	            IF #Return = TRUE THEN
	                IF #REC._FgDemArr = TRUE THEN
	                    #REC.Dial_Def.Num_Def_Etape := 1;
	                    #REC.Dial_Def.Index_Defaut := "Dialog_Defaut"(Fg_Base := #fgbase, Msg_Defaut := 'Arret immediat',
	                                                                  Type_Defaut := 2,
	                                                                  Automatisme := #REC.RecCommun.CommunGeneral._Autom,
	                                                                  Num_Lot := #REC._Ptzs._NoLot,
	                                                                  Origine_Defaut := 'Pas daction durant la suspension',
	                                                                  Libelle_Origine := 'Confirmez vous larret',
	                                                                  Acq1 := 'Confirmez',
	                                                                  Acq2 := 'Annuler',
	                                                                  Acq3 := '',
	                                                                  Acq4 := '',
	                                                                  Acq5 := '',
	                                                                  Acq6 := '',
	                                                                  Acq7 := '',
	                                                                  Acq8 := '',
	                                                                  Acq_Choisi := -1,
	                                                                  Date_Arrivee := #REC._TpsPicke);
	                    #REC.RecCommun.CommunGeneral._Etp := #Etape_Attente_RepDial;
	                    RETURN;
	                ELSE
	                    #Ret := "Arr_Imm_Circuit"(#REC._PtCir);
	                    #REC.Dial_Def.Reponse_Def := '';
	                    #REC._FgConfArret := TRUE;
	                    (* #Ret := "Arr_Imm_Circuit"(#REC._PtCir);
	                    #REC.RecCommun.CommunGeneral._Etp :=  #Etape_fin_lot; *)
	                    RETURN;
	                END_IF;
	            END_IF;
	        SUSPENSION_DEF1:
	            //======================== Traitement des reponses pour le defaut1 Etape Suspension  ====================================//
	            IF #REC.Dial_Def.Reponse_Def = 'Confirmez' THEN
	                #Ret := "Arr_Imm_Circuit"(#REC._PtCir);
	                #REC.Dial_Def.Reponse_Def := '';
	                #REC._FgConfArret := TRUE;
	                // #REC.RecCommun.CommunGeneral._Etp :=  #Etape_fin_lot;
	                RETURN;
	            END_IF;
	            IF #REC.Dial_Def.Reponse_Def = 'Annuler' THEN
	                //Renitialiser la temporisation pour refaire le test
	                #Ret_RD_Sys_T := RD_SYS_T(#REC._TpsPicke);
	                #REC.Dial_Def.Reponse_Def := '';
	                RETURN;
	            END_IF;
	            //======================================  Fin traitement====================================//
	            (* //pas de dialogue pour Confirmez l'arret
	            IF #Return AND #REC._FgDemArr = FALSE THEN
	                #Ret := "Arr_Imm_Circuit"(#REC._PtCir);
	                #REC.Dial_Def.Reponse_Def := '';
	                #REC._FgConfArret := TRUE;
	                (* #Ret := "Arr_Imm_Circuit"(#REC._PtCir);
	                #REC.RecCommun.CommunGeneral._Etp :=  #Etape_fin_lot; *)
	                RETURN;
	            END_IF; *)
	            IF (#REC._FgArret = TRUE) THEN
	                #REC._Ptzs._QteLot := #REC.RecCommun.CommunGeneral._ParCal._QteTrans;

	                "MAJ_Cumul_Dest"(Dest := "Nom_Mobile"(#REC.RecCommun.CommunGeneral._Ptdest),
	                                 Increment := FALSE,
	                                 DestR := #REC._Ptzs._DestR,
	                                 PARCAL := #REC.RecCommun.CommunGeneral._ParCal);
	                //Fin_Lot_Circuit(_ptCir, _ptCir->Origine.Mobile, _ptCir->Destination.Mobile, pt_zs->QteLot);
	                #REC.RecCommun.CommunGeneral._Etp := #Etape_maj_base;
	                RETURN;
	            END_IF;
	            IF #REC._FgSusp = FALSE THEN
	                //APPEL FCT MARCHE MOB
	                //"DB_BIBLIOTHEQUE".Mobile["DB_BIBLIOTHEQUE".Mobile[#REC._PtCir.Origine].Mob_Suiv[0]].Ord := 0; // Appl fct arrt mob
	                IF NOT #REC._FgConfArret THEN
	                    #Ret := "Dem_Mobile"("DB_BIBLIOTHEQUE".Mobile[#REC._PtCir.Origine].Mob_Suiv[0]);
	                    #REC.RecCommun.CommunGeneral._Etp := #Etape_surveillance;
	                    RETURN;
	                ELSE
	                    #REC.RecCommun.CommunGeneral._Etp := #Etape_prepositionnement;
	                    RETURN;
	                END_IF;




	            END_IF;
	            IF (#REC._FgDemVid = TRUE) THEN
	                //#REC._FgSusp := FALSE;
	                #REC.RecCommun.CommunGeneral._Etp := #Etape_vidange;
	                RETURN;
	            END_IF;


	        END_REGION Traitement cyclique "Suspension"
	        RETURN;
	(*
	 *************************************** *************************************** *************************************** *************************************** *************************************** ***************************************
	                                                                                 ╔════════════════════════════════════╗
	                                                                                 ║        Etape "Test Qte passée"     ║
	                                                                                 ╚════════════════════════════════════╝
	 *************************************** *************************************** *************************************** *************************************** *************************************** ***************************************
	*)
	    #Etape_test_qte_passee:
	        REGION Traitement preliminaire 'Test qte passee'
	            IF (#REC.RecCommun.CommunGeneral._Etp <> #REC.RecCommun.CommunGeneral._EtpPrec) THEN

	                //Memorisation de l'etape encours
	                #REC.RecCommun.CommunGeneral._EtpPrec := #REC.RecCommun.CommunGeneral._Etp;
	                //Reperer le niveau du grafcet
	                #MajNiv := "Maj_Niv"(Num_Zone := #REC.RecCommun.CommunGeneral._NumZone, Num_Tache := #REC.RecCommun.CommunGeneral._Tache, Niveau := "REC_TestQtePassee_Niv");
	                //Nomination l'etape en cours
	                #REC.RecCommun.CommunGeneral._DescEtp := 'Test qte pasee';
	                IF #REC.Dial_Def.Reponse_Def <> '' THEN
	                    CASE #REC.Dial_Def.Num_Def_Etape OF
	                        1:
	                            GOTO TEST_QTE_PASSEE_DEF1;
	                    END_CASE;
	                END_IF;
	                #Ret_RD_Sys_T := RD_SYS_T(#REC._TpsPicke);
	                #REC._DebutMax := #REC._TpsPicke;
	                IF #REC.RecCommun.CommunGeneral._ParCal._DebVolTrans = 0 OR #REC.RecCommun.CommunGeneral._ParCal._DebMasTrans = 0 OR
	                    #REC.RecCommun.CommunGeneral._ParCal._QteTrans = 0 OR #REC._TheoTrans = 0 OR #REC._SeuilTrans = 0
	                    OR #REC._FgTestQtP = FALSE THEN
	                    #REC.RecCommun.CommunGeneral._Etp := #Etape_vidange;
	                    RETURN;
	                END_IF;
	                #REC._FgAbandon := FALSE;
	            END_IF;
	        END_REGION Traitement preliminaire 'Test qte passee'

	        REGION Traitement cyclique "Test qte passee"
	            // mise a jour quantité theorique calculé en zone de suivi
	            #REC._Ptzs._Qte_Rec := #REC.RecCommun.CommunGeneral._ParCal._QteTrans;
	            // mise a jour temps de marche transporteur dans zone de suivi
	            #REC._Ptzs._Tps_Tc := #REC.RecCommun.CommunGeneral._ParCal._TpsTran;
	            //calcul debit massique
	            "Debit_Massique"(SAV := #REC._vitesseFosse,
	                             Densite := #REC._Ptzs._Densite,
	                             PARCAL := #REC.RecCommun.CommunGeneral._ParCal);
	            //test demande d'arret par bouton sur supervision
	            IF #REC._FgArret THEN
	                #REC.RecCommun.CommunGeneral._Etp := #Etape_vidange;
	                RETURN;
	            END_IF;
	            //test demande de vidange par bouton sur supervision
	            IF #REC._FgDemVid THEN
	                #REC.RecCommun.CommunGeneral._Etp := #Etape_vidange;
	                RETURN;
	            END_IF;
	            //test demande de suspension par bouton sur supervision
	            IF #REC._FgSusp THEN
	                #REC.RecCommun.CommunGeneral._Etp := #Etape_suspension;
	                RETURN;
	            END_IF;
	            //teste niveau haut
	            #Ret := "Controle_NH"(TempoAffNH := "TpDefNh", R := #REC);
	            IF #Ret = 1 THEN
	                #REC.RecCommun.CommunGeneral._Etp := #Etape_changement_destination;
	                RETURN;
	            END_IF;
	            //Controle quantité passée
	            IF #REC.RecCommun.CommunGeneral._ParCal._QteTrans >= (#REC._TheoTrans - #REC._SeuilTrans) OR #REC._FgAbandon THEN
	                IF #REC._FgAbandon = FALSE THEN
	                    #REC._Ptzs._Fg_Qte_Passee := TRUE;
	                END_IF;
	                #REC.RecCommun.CommunGeneral._Etp := #Etape_vidange;
	                RETURN;
	            END_IF;
	            //decompte tempo maxi avant dialogue de defaut
	            #Return := "Tempo"(Duree := #REC._TpMaxFPm, Tps_Picke := #REC._DebutMax, Anticip := FALSE, Tps_Passe => #Tps_Passe);
	            IF #Return AND #REC._FgAbandon = false THEN
	                #REC.Dial_Def.Num_Def_Etape := 1;
	                #REC.Dial_Def.Index_Defaut := "Dialog_Defaut"(Fg_Base := #fgbase, Msg_Defaut := 'Perte de matiere',
	                                                              Type_Defaut := 2,
	                                                              Automatisme := #REC.RecCommun.CommunGeneral._Autom,
	                                                              Num_Lot := #REC._Ptzs._NoLot,
	                                                              Origine_Defaut := 'Pas de presence du matiere',
	                                                              Libelle_Origine := 'Pas de presence du matiere',
	                                                              Acq1 := 'Relance',
	                                                              Acq2 := 'Abandon',
	                                                              Acq3 := '',
	                                                              Acq4 := '',
	                                                              Acq5 := '',
	                                                              Acq6 := '',
	                                                              Acq7 := '',
	                                                              Acq8 := '',
	                                                              Acq_Choisi := -1,
	                                                              Date_Arrivee := #REC._TpsPicke);
	                #REC.RecCommun.CommunGeneral._Etp := #Etape_Attente_RepDial;
	                RETURN;
	            END_IF;
	        TEST_QTE_PASSEE_DEF1:
	            //======================== Traitement des reponses pour le defaut1 Etape TEST QTE PASSEE Perte PM  ====================================//
	            IF #REC.Dial_Def.Reponse_Def = 'Relance' THEN //relance
	                #REC._DebutMax := #REC._TpsPicke;
	                #REC.Dial_Def.Reponse_Def := '';
	                RETURN;
	            END_IF;
	            IF #REC.Dial_Def.Reponse_Def = 'Abandon' THEN //abandon
	                #REC._FgAbandon := TRUE;
	                #REC.Dial_Def.Reponse_Def := '';
	                RETURN;
	            END_IF;
	            //======================================  Fin traitement====================================//
	        END_REGION Traitement cyclique "Test qte passee"

	        RETURN;
	(*
	 *************************************** *************************************** *************************************** *************************************** *************************************** ***************************************
	                                                                                 ╔════════════════════════════════════╗
	                                                                                 ║   Etape "Attente Acq nettoyage"    ║
	                                                                                 ╚════════════════════════════════════╝
	 *************************************** *************************************** *************************************** *************************************** *************************************** ***************************************
	*)
	    #Etape_attente_acquit_nettoyage:

	        REGION Traitement preliminaire 'Attente_acquit_nettoyage'
	            IF (#REC.RecCommun.CommunGeneral._Etp <> #REC.RecCommun.CommunGeneral._EtpPrec) THEN
	                //Memorisation de l'etape encours
	                #REC.RecCommun.CommunGeneral._EtpPrec := #REC.RecCommun.CommunGeneral._Etp;
	                //Reperer le niveau du grafcet
	                #MajNiv := "Maj_Niv"(Num_Zone := #REC.RecCommun.CommunGeneral._NumZone, Num_Tache := #REC.RecCommun.CommunGeneral._Tache, Niveau := "REC_AttenteAcquitNettoyage_Niv");
	                //Nomination l'etape en cours
	                #REC.RecCommun.CommunGeneral._DescEtp := 'Attente acquit nettoyage';
	            END_IF;
	        END_REGION Traitement preliminaire 'Attente_acquit_nettoyage'

	        REGION Traitement cyclique "Attente acquit nettoyage"

	        END_REGION Traitement cyclique "Attente acquit nettoyage"
	        RETURN;
	        RETURN;

	(*
	 *************************************** *************************************** *************************************** *************************************** *************************************** ***************************************
	                                                                                 ╔════════════════════════════════════╗
	                                                                                 ║          Etape "Vidange"           ║
	                                                                                 ╚════════════════════════════════════╝
	 *************************************** *************************************** *************************************** *************************************** *************************************** ***************************************
	*)

	    #Etape_vidange:
	        REGION Traitement preliminaire 'Vidange'

	            IF (#REC.RecCommun.CommunGeneral._Etp <> #REC.RecCommun.CommunGeneral._EtpPrec) THEN
	                #Ret_RD_Sys_T := RD_SYS_T(#REC._TpsPicke);
	                #REC._Ptzs._DateArretTC := #REC._TpsPicke;
	                //Memorisation de l'etape encours
	                #REC.RecCommun.CommunGeneral._EtpPrec := #REC.RecCommun.CommunGeneral._Etp;
	                //Reperer le niveau du grafcet
	                #MajNiv := "Maj_Niv"(Num_Zone := #REC.RecCommun.CommunGeneral._NumZone, Num_Tache := #REC.RecCommun.CommunGeneral._Tache, Niveau := "REC_Vidange_Niv");
	                //Nomination l'etape en cours
	                #REC.RecCommun.CommunGeneral._DescEtp := 'Etape Vidange';
	                #REC._FgDemVid := FALSE;

	                #REC._Ptzs._QteLot := #REC.RecCommun.CommunGeneral._ParCal._QteTrans;

	                //#REC._FgDemQteP := FALSE;
	                // #REC._FgRepQteP := FALSE;
	                #REC._FgActQtePossible := FALSE;
	                //#Ret := "Fin_Pos_Circuit"(#REC._PtCir);
	            END_IF;
	        END_REGION Traitement preliminaire 'Vidange'

	        REGION Traitement cyclique "Vidange"
	            #Ret_Bool := "Vid_Circuit_Cycl"(#REC._PtCir);
	            IF #Ret_Bool AND "Test_Etat_Circuit"(Etat := "Libre", Debut := 0, CIRCUIT := #REC._PtCir) THEN
	                // IF "Test_Etat_Circuit"(Etat := "Enc_Fin_Pos", Debut := 0, CIRCUIT := #REC._PtCir) THEN
	                #Ret := "Libere_Circuit"(#REC._PtCir);

	                "MAJ_Cumul_Dest"(Dest := "Nom_Mobile"(#REC.RecCommun.CommunGeneral._Ptdest),
	                                 Increment := FALSE,
	                                 DestR := #REC._Ptzs._DestR,
	                                 PARCAL := #REC.RecCommun.CommunGeneral._ParCal);
	                #REC._CumulQteNh := #REC._Ptzs._DestR._Liste[#REC._Ptzs._DestR._Index]._CumulQte;
	                #REC.RecCommun.CommunGeneral._Etp := #Etape_maj_base;
	            END_IF;
	        END_REGION Traitement cyclique "Vidange"


	        RETURN;
	(*
	 *************************************** *************************************** *************************************** *************************************** *************************************** *************************************** ***************************************
	                                                                                 ╔════════════════════════════════════╗
	                                                                                 ║          Etape "MAJ Base"          ║
	                                                                                 ╚════════════════════════════════════╝
	 *************************************** *************************************** *************************************** *************************************** *************************************** *************************************** ***************************************
	*)
	    #Etape_maj_base:

	        REGION Traitement preliminaire 'Maj Base'
	            IF (#REC.RecCommun.CommunGeneral._Etp <> #REC.RecCommun.CommunGeneral._EtpPrec) THEN
	                //Memorisation de l'etape encours
	                #REC.RecCommun.CommunGeneral._EtpPrec := #REC.RecCommun.CommunGeneral._Etp;
	                //Reperer le niveau du grafcet

	                #MajNiv := "Maj_Niv"(Num_Zone := #REC.RecCommun.CommunGeneral._NumZone, Num_Tache := #REC.RecCommun.CommunGeneral._Tache, Niveau := "REC_MajBase_Niv");
	                //Nomination l'etape en cours
	                #REC.RecCommun.CommunGeneral._DescEtp := 'Maj Base';
	            END_IF;
	        END_REGION Traitement preliminaire 'Maj Base'

	        REGION Traitement cyclique "Maj Base"
	            IF NOT #REC._FgAbandon THEN
	                IF #REC._FgGestDens THEN
	                    #ret_sint := "CorDensite"(QteReelle := #REC._Ptzs._Qte_Prev,
	                                              QteCalculee := #REC.RecCommun.CommunGeneral._ParCal._QteTrans,
	                                              AncCoeff := #REC._Ptzs._CoefDens,
	                                              PasMaxCorCoeff := #REC._PasMaxCorCoeff,
	                                              DensCorMax := #REC._DensMaxi,
	                                              DensCorMin := #REC._DensMini,
	                                              DensInitial := #REC._Ptzs._Densite,
	                                              TolMax := #REC._TolMax,
	                                              TolMin := #REC._TolMin,
	                                              NvCoeff := #REC._AffCoefCor,
	                                              DensCor := #REC._AffDensCours);
	                END_IF;
	                IF #fgbase AND #ret_sint = 0 THEN
	                    // Appel Proc RecrCoef Proc_RecrCoef(pt_zs->Cd_Mat,LireIdIdCoeffDens(),AnsiString(WLireProcede()).c_str(),_nouvCoef);
	                    ;
	                END_IF;


	            END_IF;




	            #REC.RecCommun.CommunGeneral._Etp := #Etape_fin_lot;
	        END_REGION Traitement cyclique "Maj Base"
	        RETURN;
	(*
	 *************************************** *************************************** *************************************** *************************************** *************************************** ***************************************
	                                                                                 ╔════════════════════════════════════╗
	                                                                                 ║          Etape "Fin Lot"           ║
	                                                                                 ╚════════════════════════════════════╝
	 *************************************** *************************************** *************************************** *************************************** *************************************** ***************************************
	*)
	    #Etape_fin_lot:
	        REGION Traitement preliminaire 'Fin Lot'
	            IF (#REC.RecCommun.CommunGeneral._Etp <> #REC.RecCommun.CommunGeneral._EtpPrec) THEN
	                //Memorisation de l'etape encours
	                #REC.RecCommun.CommunGeneral._EtpPrec := #REC.RecCommun.CommunGeneral._Etp;
	                //Nomination l'etape en cours
	                #REC.RecCommun.CommunGeneral._DescEtp := 'Fin Lot';
	                #REC._FgArret := FALSE;
	                #REC._FgActQtePossible := FALSE;
	                IF #REC.Dial_Def.Reponse_Def <> '' THEN
	                    CASE #REC.Dial_Def.Num_Def_Etape OF
	                        1:
	                            GOTO FinLot_DEF1;
	                    END_CASE;
	                END_IF;
	                // Appel fonction fn réception
	                IF #fgbase THEN
	                    #ResultProcFinRec := "Proc_Fin_Recep"(NumPoste := "Num_Poste", IdRecep := #REC._Ptzs._Id_Rec,
	                                                          CumulTps := #REC.RecCommun.CommunGeneral._ParCal._TpsTran / 1000, Msg_Def => #Text_Def);
	                    #ResultProcFinRec := 'OK';
	                ELSE
	                    #ResultProcFinRec := 'OK';
	                END_IF;


	            END_IF;
	        END_REGION Traitement preliminaire 'Fin Lot'

	        REGION Traitement cyclique "Fin Lot"
	            IF #ResultProcFinRec <> 'OK' THEN
	                #REC.Dial_Def.Num_Def_Etape := 1;
	                #REC.Dial_Def.Index_Defaut := "Dialog_Defaut"(Fg_Base := #fgbase, Msg_Defaut := #ResultProcFinRec,
	                                                              Type_Defaut := 2,
	                                                              Automatisme := #REC.RecCommun.CommunGeneral._Autom,
	                                                              Num_Lot := #REC._Ptzs._NoLot,
	                                                              Origine_Defaut := 'Base de donnees',
	                                                              Libelle_Origine := 'Base de donnees',
	                                                              Acq1 := 'Abandon',
	                                                              Acq2 := 'Relance',
	                                                              Acq3 := '',
	                                                              Acq4 := '',
	                                                              Acq5 := '',
	                                                              Acq6 := '',
	                                                              Acq7 := '',
	                                                              Acq8 := '',
	                                                              Acq_Choisi := -1,
	                                                              Date_Arrivee := #REC._TpsPicke);
	                #REC.RecCommun.CommunGeneral._Etp := #Etape_Attente_RepDial;
	                RETURN;
	            END_IF;
	        FinLot_DEF1:
	            //================================== Traitement des reponses pour le defaut1  =============================================================//
	            IF #REC.Dial_Def.Reponse_Def = 'Abandon' THEN
	                #ResultProcFinRec := 'OK';
	                #REC.Dial_Def.Reponse_Def := '';
	            END_IF;
	            IF #REC.Dial_Def.Reponse_Def = 'Relance' THEN
	                #REC.Dial_Def.Reponse_Def := '';
	                #ResultProcFinRec := "Proc_Fin_Recep"(NumPoste := "Num_Poste", IdRecep := #REC._Ptzs._Id_Rec,
	                                                      CumulTps := #REC.RecCommun.CommunGeneral._ParCal._TpsTran / 1000, Msg_Def => #Text_Def);
	            END_IF;
	            //============================================  Fin traitement  ====================================================================//
	            IF #ResultProcFinRec = 'OK' THEN
	                #MajNiv := "Maj_Niv"(Num_Zone := #REC.RecCommun.CommunGeneral._NumZone, Num_Tache := #REC.RecCommun.CommunGeneral._Tache, Niveau := "REC_FinLot_Niv");
	                #Ret := "Libere_Zone_Suiv_Lot"(Num_Zone := #REC.RecCommun.CommunGeneral._NumZone);
	                #REC.RecCommun.SUPREC.Commande._Suspension := FALSE;
	                #REC.RecCommun.SUPREC.Commande._Vidange := FALSE;
	                #REC.RecCommun.SUPREC.Commande._ArretImmediat := FALSE;
	                #REC.RecCommun.SUPREC.Commande._Depart := FALSE;
	                "Supervision"(RAZ := TRUE,
	                              REC := #REC);
	                #REC.TraitRec.Etape := 0;
	                #REC.RecCommun.CommunGeneral._Etp := #Etape_Repos;
	                RETURN;
	            END_IF;
	        END_REGION Traitement cyclique "Fin Lot"
	        RETURN;
	(*
	 *************************************** *************************************** *************************************** *************************************** *************************************** ***************************************
	                                                                                 ╔════════════════════════════════════╗
	                                                                                 ║ Etape "Attente Reponse Dialogue"   ║
	                                                                                 ╚════════════════════════════════════╝
	 *************************************** *************************************** *************************************** *************************************** *************************************** ***************************************
	*)
	    #Etape_Attente_RepDial:
	        REGION Preliminaire Attente Acquuitement
	            IF #REC.RecCommun.CommunGeneral._Etp <> #REC.RecCommun.CommunGeneral._EtpPrec THEN
	                //Memorisation de l'etape encours
	                #REC.RecCommun.CommunGeneral._EtpMemo := #REC.RecCommun.CommunGeneral._EtpPrec;

	                #REC.RecCommun.CommunGeneral._DescEtp := 'Etape_Attente_RepDial';
	                #REC.RecCommun.CommunGeneral._EtpPrec := #REC.RecCommun.CommunGeneral._Etp;

	            END_IF;
	        END_REGION Preliminaire Attente Acquuitement
	        REGION Cyclique Attente Acquitement
	            #REC.Dial_Def.Reponse_Def := "FC_Recup_Rep_Def"(Index_Def := #REC.Dial_Def.Index_Defaut, Reponse_Ecrit => #REC.Dial_Def.Text_Reponse);
	            IF #REC.Dial_Def.Reponse_Def <> '' THEN
	                "FC_Raz_Def"(#REC.Dial_Def.Index_Defaut);
	                #REC.RecCommun.CommunGeneral._Etp := #REC.RecCommun.CommunGeneral._EtpMemo;
	                RETURN;
	            END_IF;
	        END_REGION Cyclique Attente Acquitement
	END_CASE;

END_FUNCTION

